{attribute addProperty BoxType "EK1100-0000-0018"}
{attribute addProperty Id "Beckhoff_BKxxxxEK1122Beckhoff_BKxxxxEK1122_F2DB5C0900A_0015_BK1250_0000_0016A_0015_BK1250_0000_0016_69F539FC00"}
{attribute addProperty CRC "1700471601"}
{attribute addProperty SizeInBites "0"}
{attribute addProperty SizeInBytes "0"}
TYPE Beckhoff_BKxxxx_655B2331 EXTENDS EK1100_179A0949 :
STRUCT
	{attribute addProperty Name "Beckhoff_BKxxxxEK1122"}
	Beckhoff_BKxxxxEK1122 : Beckhoff_BKxxxxEK1122_F2DB5C09;
	{attribute addProperty Name "A_0015_BK1250_0000_0016"}
	A_0015_BK1250_0000_0016 : A_0015_BK1250_0000_0016_69F539FC;
END_STRUCT
END_TYPE

(* stored: Version 1.2.0.0, ProductVersion 3.1.4024.9
   DUT Beckhoff_BKxxxx_655B2331: Id {3a584a6a-f43e-4845-a227-4a5b1358a50e} *)
